Staubli VAL3: MFX_ROB_17.dtx

public bool bCubeStep1
public bool bCylinderStep1
bool bESTOPactive
public bool bEnableMonitor
public bool bInsideCube
public bool bInsideCylinder
public bool bInsideSphere
bool bKillRemControl
bool bMoveLinear = true
public bool bRemControlON
bool bRemMotionBusy
public bool bSetCubeXYZ
public bool bSetCylinderRZ
public bool bSetSphereRad
bool bSimESTOPOn
bool bSimulateESTOP
public bool bSphereStep1
public bool bStopAllMonitor = true
public bool bStopMotion
public bool bWatchForHalt
public bool bWorldFrameView = true
dio dCollisionSens = {link=usrIn0}
frame fIP1 = {fatherId=fIPoriginal[0]}
public frame fIP2 = {fatherId=fIPoriginal[0]}
frame fIPoriginal = {x=-1.16, y=-7.997692, z=1599.75028, rx=-90.079848, ry=0.325339, rz=-0.147005, fatherId=world[0]}
public jointRx jPark = {j1=89.588014, j2=-47.40785, j3=113.936199, j4=-0.155325, j5=-66.458795, j6=0.148711}
jointRx jParkTop = {j1=88.830052, j2=-90.553253, j3=149.996753, j4=-0.166481, j5=-59.375003, j6=0.928419}
mdesc mDefault = {accel=20, vel=20, decel=20, blend=off}
public mdesc mGlobalSpeed = {accel=20, vel=20, decel=20, blend=off}
mdesc mMdesc
public mdesc mSafeSlow = {accel=15, vel=20, decel=15, blend=off}
num nAccFast = 60
num nAccMedium = 40
num nAccSlow = 20
num nAdjPntMoveTol = 25
num nAzHere = -1.83783E-05
num nColision = 1
num nDistXCube
num nDistYCube
num nDistZCube
num nDistZCylinder
num nElHere = 44.997695
num nErrBufferSize = 10
num nErrNext
num nErrNow
num nHeartbeat = 4344
num nIP1Azimuth[20]
  [1] = 45
  [2] = -45
  [3] = 45
  [4] = -45
  [5] = 9.38
  [6] = 7.44
  [7] = 17.53
  [8] = 48.36
  [9] = 142.53
  [10] = 140.2
  [11] = 145.08
  [12] = 142.4
  [13] = 142.23
  [14] = 144.96
  [15] = 106.35
  [16] = 100.36
  [17] = 19.8
  [18] = 8.88
  [19] = 23.034688
num nIP1Elevation[20]
  [3] = -45
  [4] = -45
  [5] = 21.19
  [6] = 39.23
  [9] = 37.74
  [10] = 30.33
  [11] = 44.59
  [12] = 42.45
  [13] = 38.39
  [14] = 44.81
  [15] = 29.56
  [16] = 45.35
  [17] = 29.88
  [18] = 12.25
  [19] = 8.727177
num nIP1Number = 1
num nIP1Radius[20]
  [1] = 600
  [2] = 600
  [3] = 600
  [4] = 600
  [5] = 1000
  [6] = 1000
  [7] = 300
  [8] = 250
  [9] = 300
  [10] = 300
  [11] = 300
  [12] = 300
  [13] = 300
  [14] = 300
  [15] = 300
  [16] = 300
  [17] = 100
  [18] = 200
  [19] = 857.27654
num nIP2Azimuth[20]
  [0] = 15
  [2] = -128.927
num nIP2Elevation[20]
  [0] = 20
  [2] = 79.165
num nIP2Number = 2
num nIP2Radius[20]
  [0] = 300
  [1] = 600
  [2] = 123.321
  [5] = 1000
num nIPNumber
num nIdxAdjTargetPt = 291
num nIdxArmCalCheck = 31
num nIdxArmPowerOn = 181
num nIdxESTOPCheck = 121
num nIdxEnterIP = 341
num nIdxEnterTCP = 321
public num nIdxFrm1of5 = 131
public num nIdxFrm2of5 = 141
public num nIdxFrm3of5 = 151
public num nIdxFrm4of5 = 161
public num nIdxFrm5of5 = 171
num nIdxGetTCP = 351
public num nIdxMainMenu = 1
public num nIdxMotionMenu = 271
num nIdxMoveTargPt = 281
num nIdxMoveToPark = 311
num nIdxParkCheck = 41
public num nIdxPtrVerify
num nIdxRemControl = 321
public num nIdxResolution
public num nIdxSetCubeXYZ = 211
public num nIdxSetCylRZ = 231
num nIdxSetSpeeds = 181
public num nIdxSetSphRad = 251
num nIdxSetTargetPt = 261
public num nIdxStyClr = 61
public num nIdxTCP1of4 = 81
public num nIdxTCP2of4 = 91
public num nIdxTCP3of4 = 101
public num nIdxTCP4Point
public num nIdxTCP4of4 = 111
public num nIdxTeachClear
public num nIdxTeachCube = 201
public num nIdxTeachCyl = 221
num nIdxTeachIP = 331
public num nIdxTeachMenu = 11
public num nIdxTeachPARK = 51
num nIdxTeachPARKT = 371
public num nIdxTeachSph = 241
public num nIdxTeachTCP = 21
num nIdxUtilMenu2 = 301
num nIdxUtilityMenu = 71
num nMaxAccel = 50
num nMaxDist = 1000
num nMaxLoginTries = 3
num nMaxRVelo = 20
num nMaxVelo = 100
num nMovArgs
num nNumberCube
num nNumberCylinder
num nNumberSphere
num nPPS
num nParkTolerance = 50
num nRHere = 565.684578
num nRXHere = 0.0101053
num nRYHere = 0.000281961
num nRZHere = 0.00483895
num nRadiusCylinder
num nRadiusSphere
num nRemoteTimeout = 30
num nResolution[4]
  [0] = 0.001
  [1] = 0.01
  [2] = 0.1
  [3] = 1
num nRobotMode = 1
num nSelection = 1
num nStagePos
num nStagePosOK
num nVelFast = 60
num nVelMedium = 40
num nVelSlow = 20
num nXHere = -0.00012746
num nYHere = 399.983479
num nZHere = 400.0163407
num nZoneWatchTol = 25
public pointRx pCellReference = {shoulder=righty, elbow=epositive, wrist=wpositive, fatherId=world[0]}
pointRx pIP1NullPoint = {shoulder=sfree, elbow=efree, wrist=wfree, fatherId=fIP1[0]}
pointRx pIP1Point[20]
  [0] = {x=73, y=424, z=417, rx=-45, ry=-172, rz=-7, shoulder=sfree, elbow=efree, wrist=wfree, fatherId=fIP1[0]}
  [1] = {x=145, y=424, z=398, rx=-46, ry=-166, rz=-14, shoulder=sfree, elbow=efree, wrist=wfree, fatherId=fIP1[0]}
  [2] = {x=272, y=424, z=325, rx=-52, ry=-152, rz=-30, shoulder=sfree, elbow=efree, wrist=wfree, fatherId=fIP1[0]}
  [3] = {x=325, y=424, z=272, rx=-57, ry=-147, rz=-40, shoulder=sfree, elbow=efree, wrist=wfree, fatherId=fIP1[0]}
  [4] = {x=294, y=424, z=305, rx=-54, ry=-150, rz=-34, shoulder=sfree, elbow=efree, wrist=wfree, fatherId=fIP1[0]}
  [5] = {fatherId=fIP1[0]}
  [6] = {fatherId=fIP1[0]}
  [7] = {x=145, y=424, z=398, rx=-46, ry=-166, rz=-14, fatherId=fIP1[0]}
  [8] = {fatherId=fIP1[0]}
  [9] = {x=272, y=424, z=325, rx=-52, ry=-152, rz=-30, fatherId=fIP1[0]}
  [10] = {fatherId=fIP1[0]}
  [11] = {fatherId=fIP1[0]}
  [12] = {x=325, y=424, z=272, rx=-57, ry=-147, rz=-40, fatherId=fIP1[0]}
  [13] = {x=294, y=424, z=305, rx=-54, ry=-150, rz=-34, fatherId=fIP1[0]}
  [14] = {fatherId=fIP1[0]}
  [15] = {fatherId=fIP1[0]}
  [16] = {fatherId=fIP1[0]}
  [17] = {fatherId=fIP1[0]}
  [18] = {fatherId=fIP1[0]}
  [19] = {y=500, rx=90, rz=-180, fatherId=fIP1[0]}
pointRx pIP2NullPoint = {fatherId=fIP2[0]}
pointRx pIP2Point[20]
  [0] = {shoulder=sfree, elbow=efree, wrist=wfree, fatherId=fIP2[0]}
  [1] = {x=300, y=424.264069, z=300, rx=125.26439, ry=-30, rz=-35.26439, shoulder=sfree, elbow=efree, wrist=wfree, fatherId=fIP2[0]}
  [2] = {x=-300, y=424.264069, z=300, rx=125.26439, ry=30, rz=35.26439, shoulder=sfree, elbow=efree, wrist=wfree, fatherId=fIP2[0]}
  [3] = {x=300, y=-424.264069, z=300, rx=-125.26439, ry=-30, rz=35.26439, shoulder=sfree, elbow=efree, wrist=wfree, fatherId=fIP2[0]}
  [4] = {x=-300, y=-424.264069, z=300, rx=-125.26439, ry=30, rz=-35.26439, shoulder=sfree, elbow=efree, wrist=wfree, fatherId=fIP2[0]}
  [5] = {shoulder=sfree, elbow=efree, wrist=wfree, fatherId=fIP2[0]}
  [6] = {shoulder=sfree, elbow=efree, wrist=wfree, fatherId=fIP2[0]}
  [7] = {shoulder=sfree, elbow=efree, wrist=wfree, fatherId=fIP2[0]}
  [8] = {shoulder=sfree, elbow=efree, wrist=wfree, fatherId=fIP2[0]}
  [9] = {shoulder=sfree, elbow=efree, wrist=wfree, fatherId=fIP2[0]}
  [10] = {shoulder=sfree, elbow=efree, wrist=wfree, fatherId=fIP2[0]}
  [11] = {shoulder=sfree, elbow=efree, wrist=wfree, fatherId=fIP2[0]}
  [12] = {shoulder=sfree, elbow=efree, wrist=wfree, fatherId=fIP2[0]}
  [13] = {shoulder=sfree, elbow=efree, wrist=wfree, fatherId=fIP2[0]}
  [14] = {shoulder=sfree, elbow=efree, wrist=wfree, fatherId=fIP2[0]}
  [15] = {shoulder=sfree, elbow=efree, wrist=wfree, fatherId=fIP2[0]}
  [16] = {shoulder=sfree, elbow=efree, wrist=wfree, fatherId=fIP2[0]}
  [17] = {shoulder=sfree, elbow=efree, wrist=wfree, fatherId=fIP2[0]}
  [18] = {shoulder=sfree, elbow=efree, wrist=wfree, fatherId=fIP2[0]}
  [19] = {shoulder=sfree, elbow=efree, wrist=wfree, fatherId=fIP2[0]}
pointRx pMoveIP1Target = {fatherId=fIP1[0]}
pointRx pMoveIP2Target = {shoulder=sfree, elbow=efree, wrist=wfree, fatherId=fIP2[0]}
pointRx pMoveTarget = {shoulder=sfree, elbow=efree, wrist=wfree, fatherId=world[0]}
pointRx pNullPosition = {fatherId=world[0]}
pointRx pOriginCube = {fatherId=world[0]}
pointRx pOriginCylinder = {fatherId=world[0]}
pointRx pOriginSphere = {fatherId=world[0]}
pointRx teste[4]
  [0] = {x=7, y=243, z=26, rx=-4.03658E-18, ry=-79, rz=-9.47474E-33, shoulder=sfree, elbow=efree, wrist=wfree, fatherId=fIP1[0]}
  [1] = {x=17, y=243, z=28, rx=4.437099E-14, ry=-79.999286, rz=0.00497464, fatherId=fIP1[0]}
  [2] = {y=400, z=400, rx=0.01, ry=-2.827901E-23, rz=0.00516647, fatherId=fIP1[0]}
  [3] = {fatherId=fIP1[0]}
sio sioIOCclient = {link=Socket\MFX}
string sErrBuffer[10]
string sIOCCommand
string sIOCPassword = "USERPASSWORD"
string sIOCUserName = "CS8LOGIN"
string sIOCValue
string sIP1TargName[20]
  [0] = "v"
  [1] = "a"
  [2] = "sto 1"
  [3] = "ybco104"
  [4] = "cool oi"
  [5] = "magpeak2"
  [6] = "IP1 Point6 Name"
  [7] = "IP1 Point7 Name"
  [8] = "IP1 Point8 Name"
  [9] = "IP1 Point9 Name"
  [10] = "IP1 Point10 Name"
  [11] = "IP1 Point11 Name"
  [12] = "IP1 Point12 Name"
  [13] = "IP1 Point13 Name"
  [14] = "IP1 Point14 Name"
  [15] = "IP1 Point15 Name"
  [16] = "IP1 Point16 Name"
  [17] = "IP1 Point17 Name"
  [18] = "IP1 Point18 Name"
  [19] = "IP1 Point19 Name"
string sIP2TargName[20]
  [0] = "TestTeachPoint0"
  [1] = "IP2 Point1 Name"
  [2] = "IP2 Point2 Name"
  [3] = "IP2 Point3 Name"
  [4] = "IP2 Point4 Name"
  [5] = "a"
  [6] = "IP2 Point6 Name"
  [7] = "IP2 Point7 Name"
  [8] = "IP2 Point8 Name"
  [9] = "IP2 Point9 Name"
  [10] = "IP2 Point10 Name"
  [11] = "IP2 Point11 Name"
  [12] = "IP2 Point12 Name"
  [13] = "IP2 Point13 Name"
  [14] = "IP2 Point14 Name"
  [15] = "IP2 Point15 Name"
  [16] = "IP2 Point16 Name"
  [17] = "IP2 Point17 Name"
  [18] = "IP2 Point18 Name"
  [19] = "IP2 Point19 Name"
string sMenuBottomLine[53]
  [0] = " Tch. Mot. Util ---- ---- ---- ---- Stop"
  [1] = " Pnts IPCS Park ParkT TCP Zone  --- Ret."
  [2] = "RefP 4Pnt DEnt ---- ---- ---- ---- Ret."
  [3] = "---- ---- ---- Stop ---- ---- ---- Ret."
  [4] = "Cont ---- ---- Mov. ---- ---- ---- Ret."
  [5] = "Save ---- ---- ---- ---- ---- ---- Ret."
  [6] = "Cube Cyl. Sph. ---- ---- ---- ---- Ret."
  [7] = "Init Park Enbl Spds RemC TCP. ---- Ret."
  [8] = "Next ---- ---- ---- ---- ---- ---- Abrt"
  [9] = "Next ---- ---- ---- ---- ---- ---- Abrt"
  [10] = "Next ---- ---- ---- ---- ---- ---- Abrt"
  [11] = "Tch. ---- ---- ---- ---- ---- ---- Abrt"
  [12] = "Cont ---- ---- ---- ---- ---- ---- Abrt"
  [13] = "Next ---- Togl ---- ---- ---- ---- Abrt"
  [14] = "Next ---- ---- ---- ---- ---- ---- Abrt"
  [15] = "Next ---- ---- ---- ---- ---- ---- Abrt"
  [16] = "Next ---- ---- ---- ---- ---- ---- Abrt"
  [17] = "Save ---- ---- ---- ---- ---- ---- Abrt"
  [18] = "SVel MVel FVel ---- SAcc MAcc FAcc Ret."
  [20] = "Save ---- Chng Orig  XYZ ---- Clr. Ret."
  [21] = "Save ---- ----  DX   DY   DZ  ---- Ret."
  [22] = "Save ---- Chng Orig RadZ ---- Clr. Ret."
  [23] = "Save ---- ---- Rad.  DZ  ---- ---- Ret."
  [24] = "Save ---- Chng Orig Rad. ---- Clr. Ret."
  [25] = "Save ---- ---- Rad. ---- ---- ---- Ret."
  [26] = " IP  Pnt# Name Azi. Elev Rad.      Ret."
  [27] = "Pnts ---- ---- Park --- ParkTop -- Ret."
  [28] = " IP  Pnt# ---- ---- Adj. Mov. ---- Ret."
  [30] = "Init Park Dis. Spds RemC ---- ---- Ret."
  [31] = "Mov. ---- ---- ---- ---- ---- ---- Ret."
  [32] = " X    Y    Z    RX   RY   RZ  ---- Ret."
  [33] = "Sel. DEnt Wiz. ---- ---- ---- ---- Ret."
  [34] = " X    Y    Z    RX   RY   RZ  ---- Ret."
  [35] = " IP  ---- ---- ---- ---- ---- ---- Ret."
  [36] = "Cont ---- ---- ---- ---- ---- ---- Dis."
  [37] = "Save ---- ---- ---- ---- ---- ---- Ret."
string sNumConv = ".3"
string sRemMotionCmd
string sTargetChoice[2]
  [0] = "InteractionPoint1"
  [1] = "InteractionPoint2"
public string sUserPageText[382]
  [0] = "(F1) (F2) (F3) (F4) (F5) (F6) (F7) (F8)"
  [1] = ">>  MAIN MENU  <<"
  [2] = "Select Your Choice...     (ESC aborts)"
  [3] = "TEACH MENU"
  [4] = "MOTION MENU"
  [5] = "UTILITY MENU"
  [10] = "END PROGRAM"
  [11] = ">>  TEACH MENU  <<"
  [12] = "Select Your Choice...     (ESC aborts)"
  [13] = "Teach TARGET POINTS"
  [14] = "Teach INTERACTION PNT COORD SYS"
  [15] = "Teach PARK Position"
  [16] = "Teach PARK TOP Position"
  [17] = "Teach TCP"
  [18] = "Teach STAY CLEAR ZONES"
  [20] = "RETURN"
  [21] = ">>  TEACH TCP  <<"
  [22] = "Select Your Choice...     (ESC aborts)"
  [23] = "Teach TCP w/ REF POINTER"
  [24] = "Teach TCP w/ 4-POINT METHOD"
  [25] = "TCP Values Direct Entry"
  [30] = "ABORT & RETURN"
  [31] = ">>  ARM NOT CALIBRATED!  <<"
  [32] = "MOTION NOT ALLOWED"
  [36] = "STOP PROGRAM"
  [40] = "ABORT & RETURN"
  [41] = ">>  VERIFY ARM AT PARK <<"
  [42] = "Select Your Choice...     (ESC aborts)"
  [46] = "Move to PARK"
  [50] = "ABORT & RETURN"
  [51] = ">>  TEACH PARK Position  <<"
  [52] = "               (ESC aborts)"
  [53] = "Instructions:"
  [54] = "1.  Change to MANUAL mode"
  [55] = "2.  Move robot to  PARK location"
  [59] = "(F1)  ACCEPT, SAVE, & RETURN"
  [60] = "(F8)  ABORT & RETURN"
  [61] = ">>  DEFINE STAY CLEAR ZONES  <<"
  [62] = "Select Your Choice...     (ESC aborts)"
  [63] = "CUBE Zones"
  [64] = "CYLINDER Zones"
  [65] = "SPHERE Zones"
  [70] = "ABORT & RETURN"
  [71] = ">>  UTILITY MENU  <<"
  [72] = "Select Your Choice...     (ESC aborts)"
  [73] = "Initialize Robot"
  [74] = "Verify Arm is at PARK location"
  [75] = "ENABLE  Zone Monitoring"
  [76] = "Set Global Speed Parameters"
  [77] = "Start IOC Client Remote Control"
  [78] = "Show Current TCP:IP Frame Vals"
  [80] = "RETURN"
  [81] = ">> TEACH TCP w/ Pointer:  1 of 4  <<"
  [82] = "               (ESC aborts)"
  [83] = "CONDITIONS REQD TO TEACH TCP"
  [84] = "#1:  Ref Pointer attached to Flange"
  [85] = "    (Defined tool = tRefPointer)"
  [86] = "#2:  Cell Ref Pointer in Workspace"
  [89] = "(F1)  CONTINUE to Step 2 of 4"
  [90] = "(F8)  ABORT & RETURN"
  [91] = ">>  TEACH TCP w/ Pointer:  2 of 4  <<"
  [92] = "               (ESC aborts)"
  [94] = "          MOVE ROBOT TO"
  [95] = "     CELL REFERENCE POINTER"
  [99] = "(F1)  CONTINUE to Step 3 of 4"
  [100] = "(F8)  ABORT & RETURN"
  [101] = ">>  TEACH TCP w/ Pointer:  3 of 4  <<"
  [102] = "               (ESC aborts)"
  [103] = "       DO THE FOLLOWING"
  [104] = "1.  REMOVE Reference Pointer Tool"
  [105] = "2.  ATTACH Sensor Tool"
  [106] = "3.  MOVE Sensor Tool to Cell Ref Ptr"
  [109] = "(F1) TEACH TOOL & CONTINUE"
  [110] = "(F8) ABORT & RETURN"
  [111] = ">>  TEACH TCP w/ Pointer:  4 of 4  <<"
  [112] = "               (ESC aborts)"
  [113] = "VERIFY the Sensor Tool Definition:"
  [114] = "1.  Switch to TOOL MODE on Pendant"
  [115] = "2.  Move  X, Y, Z, RX, RY, RZ "
  [116] = "  and verify motion"
  [119] = "(F1)  ACCEPT, SAVE,  AND RETURN"
  [120] = "(F8)  ABORT & RETURN WITHOUT SAVE"
  [121] = ">>  ESTOP CHECK <<"
  [122] = "Select Your Choice...     (ESC aborts)"
  [123] = "(F1)  Continue"
  [130] = "(F8)  ABORT & RETURN"
  [131] = ">>  TEACH IP COORD SYS:  1 of 5  <<"
  [132] = "               (ESC aborts)"
  [134] = "SELECT IP COORD SYS TO TEACH"
  [136] = "(F1)  ACCEPT & CONTINUE"
  [138] = "(F3)  Toggle INT POINT CS Selection"
  [140] = "(F8)  ABORT & RETURN"
  [141] = ">>  TEACH INT POINT CS:  2 of 5  <<"
  [142] = "               (ESC aborts)"
  [145] = "ATTACH REF POINTER"
  [146] = "TO ROBOT FLANGE"
  [149] = "(F1)  CONTINUE"
  [150] = "(F8)  ABORT & RETURN"
  [151] = ">>  TEACH INT POINT CS:  3 of 5  <<"
  [152] = "               (ESC aborts)"
  [155] = "MOVE  REF POINTER TO"
  [156] = "INTERATION POINT COORD SYS"
  [157] = "ORIGIN POINT"
  [159] = "(F1)  CONTINUE"
  [160] = "(F8)  ABORT & RETURN"
  [161] = ">>  TEACH INT POINT CS:  4 of 5  <<"
  [162] = "               (ESC aborts)"
  [165] = "MOVE REF POINTER TO"
  [166] = "INTERACTION POINT COORD SYS"
  [167] = "X-AXIS POINT"
  [169] = "(F1)  CONTINUE"
  [170] = "(F8)  ABORT & RETURN"
  [171] = ">>  TEACH INT POINT CS:  5 of 5  <<"
  [172] = "               (ESC aborts)"
  [175] = "MOVE REF POINTER TO"
  [176] = "INTERACTION POINT COORD SYS"
  [177] = "Y-AXIS POINT"
  [179] = "(F1)  ACCEPT, SAVE,  & RETURN"
  [180] = "(F8)  ABORT & RETURN WITHOUT SAVE"
  [181] = ">>  SET GLOBAL SPEED PARMS  <<"
  [182] = "Select Your Choice...     (ESC aborts)"
  [183] = "Slow Speed"
  [184] = "Medium Speed"
  [185] = "Fast Speed"
  [187] = "Slow Accel"
  [188] = "Medium Accel"
  [189] = "Fast Accel"
  [190] = "Return"
  [191] = ">>  TEACH PARK Position  <<"
  [192] = "               (ESC aborts)"
  [193] = "Move to PARK Position, F1 to continue..."
  [200] = "GO BACK"
  [201] = ">>  DEFINE CUBE Stay Clear Zone  <<"
  [202] = "               (ESC aborts)"
  [204] = "(F1)  ACCEPT, SAVE, & RETURN"
  [206] = "(F3)  Change Cube Number"
  [207] = "(F4)  Teach Cube Origin Point"
  [208] = "(F5)  Define DX, DY, DZ"
  [209] = "(F7)  Clear This Cube Definition"
  [210] = "(F8)  ABORT & RETURN"
  [211] = ">>  SET CUBE DX DY DZ <<"
  [212] = "               (ESC aborts)"
  [215] = "(F1)  ACCEPT DX/DY/DZ VALUES"
  [216] = "(F4)  Enter New DX Value"
  [217] = "(F5)  Enter New DY Value"
  [218] = "(F6)  Enter New DZ Value"
  [220] = "(F8)  ABORT & RETURN"
  [221] = ">>  DEFINE CYLINDER Stay Clear Zone  <<"
  [222] = "               (ESC aborts)"
  [224] = "(F1)  ACCEPT, SAVE, & RETURN"
  [226] = "(F3)  Change Cylinder Number"
  [227] = "(F4)  Teach Cylinder Origin Point"
  [228] = "(F5)  Define Cylinder Radius & DZ"
  [229] = "(F7)  Clear this Cylinder Definition"
  [230] = "(F8)  ABORT & RETURN"
  [231] = ">>  SET CYLINDER RAD & DZ  <<"
  [232] = "               (ESC aborts)"
  [235] = "(F1)  ACCEPT RAD/DZ VALUES"
  [236] = "(F4)  Enter New RADIUS Value"
  [237] = "(F5)  Enter New DZ Value"
  [240] = "(F8)  ABORT & RETURN"
  [241] = ">>  DEFINE SPHERE Stay Clear Zone  <<"
  [242] = "               (ESC aborts)"
  [244] = "(F1)  ACCEPT, SAVE, & RETURN"
  [246] = "(F3)  Change Sphere Number"
  [247] = "(F4)  Teach Sphere Origin Point"
  [248] = "(F5)  Define Sphere Radius"
  [249] = "(F7)  Clear This Sphere Definition"
  [250] = "(F8)  ABORT & RETURN"
  [251] = ">>  SET SPHERE RADIUS  <<"
  [252] = "               (ESC aborts)"
  [255] = "(F1)  ACCEPT RADIUS VALUE"
  [256] = "(F4)  Enter New RADIUS Value"
  [260] = "(F8)  ABORT & RETURN"
  [261] = ">>  SET TARGET POINTS  <<"
  [262] = "(F1) IP Nbr      :"
  [263] = "(F2) Pnt Nbr     :"
  [264] = "(F3) Name        :"
  [265] = "(F4) Azimuth     :"
  [266] = "(F5) Elevation   :"
  [267] = "(F6) Radius      :"
  [268] = "     X:         Y:         Z:"
  [269] = "    RX:        RY:        RZ:"
  [270] = "(F8)  SAVE, UPDATE, & RETURN"
  [271] = ">>  MOTION MENU  <<"
  [272] = "Select Your Choice...     (ESC aborts)"
  [273] = "Move & Adjust TARGET POINTS"
  [276] = "Move to PARK POSITION"
  [278] = "Move to PARK TOP POSITION"
  [280] = "ABORT"
  [281] = ">>  MOVE & ADJUST TARGET POINTS  <<"
  [282] = "(F1) IP Nbr      :"
  [283] = "(F2) Pnt Nbr     :"
  [284] = "        Name        :"
  [285] = "       Azimuth     :"
  [286] = "       Elevation   :"
  [287] = "       Radius      :"
  [288] = "     X:         Y:         Z:"
  [289] = "    RX:        RY:        RZ:"
  [290] = "(F6) MOVE TO   (F8) ABORT & RETURN"
  [291] = ">>  ADJUST TARGET POINTS  <<"
  [296] = "  Resolution:"
  [297] = "  Target RX:"
  [298] = "  Target RY:"
  [299] = "  Target RZ:"
  [301] = ">>  UTILITY MENU  <<"
  [302] = "Select Your Choice...     (ESC aborts)"
  [303] = "Initialize Robot"
  [304] = "Verify Arm is at PARK location"
  [305] = "DISABLE Zone Monitoring"
  [306] = "Set Global Speed Parameters"
  [307] = "Start IOC Host Remote Control"
  [310] = "RETURN"
  [311] = ">>  MOVE TO  PARK  <<"
  [312] = "Select Your Choice...     (ESC aborts)"
  [313] = "Start Move to PARK Location"
  [320] = "ABORT"
  [321] = ">>  DIRECT ENTRY TCP VALUES  <<"
  [322] = " Enter Values...        ESC Aborts"
  [323] = " TCP-X"
  [324] = " TCP-Y"
  [325] = " TCP-Z"
  [326] = " TCP-RX"
  [327] = " TCP-RY"
  [328] = " TCP-RZ"
  [330] = " F8 = Save & Return"
  [331] = ">> TEACH INTERATION PNTS <<"
  [332] = "Select Your Choice...       ESC Aborts"
  [333] = "(F1)  Select Interaction Point"
  [334] = "(F2)  Direct Entry of IP Data"
  [335] = "(F3)  Run IP Teach Wizard"
  [337] = "(F8)  Return"
  [341] = ">>  DIRECT ENTRY IP VALUES  <<"
  [342] = " Enter Values...        ESC Aborts"
  [343] = "IP-X"
  [344] = "IP-Y"
  [345] = "IP-Z"
  [346] = "IP-RX"
  [347] = "IP-RY"
  [348] = "IP-RZ"
  [350] = "(F8)  Save & Return"
  [351] = ">>  DISPLAY TCP VALUES @ IP  <<"
  [352] = "                        ESC Aborts"
  [353] = "Current IP  :"
  [354] = "TCP.x       :"
  [355] = "TCP.y       :"
  [356] = "TCP.z       :"
  [357] = "TCP.rx      :"
  [358] = "TCP.ry      :"
  [359] = "TCP.rz      :"
  [361] = ">>  STARTUP CHECK 0UT  <<"
  [363] = "WARNING:  ESTOP Simulation = ACTIVE !"
  [365] = "F1:  CONTINUE"
  [367] = "F8:  Disable ESTOP Simulation"
  [370] = "ABORT & RETURN"
  [371] = ">>  TEACH PARK Position  <<"
  [372] = "               (ESC aborts)"
  [373] = "Instructions:"
  [374] = "1.  Change to MANUAL mode"
  [375] = "2.  Move robot to  PARK TOP location"
tool tNULLTOOL = {fatherId=flange[0], ioLink=valve1}
public tool tRefPointer = {fatherId=flange[0], ioLink=valve1}
tool tSensorTool = {z=162.433, ry=90, rz=-90, fatherId=flange[0], ioLink=valve1}
trsf trUserTool
